FUNCTION_BLOCK LOAD_CSV_SIM
  {SET_ATTRIBUTE(OpcUa, DEVICE.SENSOR)}
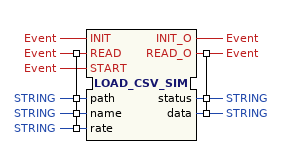
  EVENT_INPUT
    INIT;
    READ WITH path, name, rate; {SET_ATTRIBUTE(OpcUa, Method)}
    START;
  END_EVENT
  EVENT_OUTPUT
    INIT_O;
    READ_O WITH status, data;
  END_EVENT
  VAR_INPUT
    path : STRING; {SET_ATTRIBUTE(OpcUa, Constant)}
    name : STRING; {SET_ATTRIBUTE(OpcUa, Constant)}
    rate : STRING; {SET_ATTRIBUTE(OpcUa, Constant)}
  END_VAR
  VAR_OUTPUT
    status : STRING; {SET_ATTRIBUTE(OpcUa, Variable)}
    data : STRING; {SET_ATTRIBUTE(OpcUa, Variable)}
  END_VAR
END_FUNCTION_BLOCK
